// TwinCAT 3 PLC project Library_OOP
// Title: Library_OOP_Course
// Company: Course_OOP
// Author: Victor Duran -- Runtimevic
// ProjectVersion: 0.0.0.2
// Description: Library Couse OOP
// ProgramVersion: 3.1.4024.0
// libraries:
//   Library_OOP_Course, * (Course_OOP)
//   Tc2_Standard, * (Beckhoff Automation GmbH)
//   Tc2_System, * (Beckhoff Automation GmbH)
//   Tc3_Module, * (Beckhoff Automation GmbH)
// project tree:
//   Components/Cylinder/Interfaces/ I_AtHome.TcIO (not stored), I_AtWork.TcIO (not stored), I_MoveTo.TcIO (not stored)
//   FBs/ FB_FB_AXL_E_EC_DI8_DO8_M12_6P_BitMaps.TcPOU
//   FCs/ FC_Sum_int.TcPOU, FC_Word2Bools.TcPOU
//   / PlcTask.TcTTO
//   POUs/ MAIN.TcPOU
//   Project Information/ F_GetCompany.TcPOU, F_GetTitle.TcPOU, F_GetVersion.TcPOU
//   Units/DigitalInput/Class/ FB_DigitalInput.TcPOU (not stored)
//   Units/DigitalInput/Interface/ I_DigitalStatus.TcIO (not stored)
//   Units/DigitalOutput/Class/ FB_DigitalOutput.TcPOU (not stored)
//   Units/DigitalOutput/Interface/ I_DigitalOutput.TcIO (not stored)
//   Version/ Global_Version.TcGVL
// real-time tasks:
//   TASK PlcTask: cycle T#10ms, priority 20, ADS port 350

CONFIGURATION Library_OOP
    RESOURCE PLC ON TwinCAT3
        TASK PlcTask(INTERVAL := T#10ms, PRIORITY := 20);
        PROGRAM MAIN WITH PlcTask : MAIN;
    END_RESOURCE
END_CONFIGURATION

// ---- Version/Global_Version.TcGVL
{attribute 'TcGenerated'}
{attribute 'no-analysis'}
{attribute 'linkalways'}
// This function has been automatically generated from the project information.
VAR_GLOBAL CONSTANT
	{attribute 'const_non_replaced'}
	stLibVersion_Library_OOP_Course : ST_LibVersion := (iMajor := 0, iMinor := 0, iBuild := 0, iRevision := 2, nFlags := 1, sVersion := '0.0.0.2');
END_VAR

// ---- POUs/MAIN.TcPOU
PROGRAM MAIN
VAR
END_VAR

END_PROGRAM

// ---- FBs/FB_FB_AXL_E_EC_DI8_DO8_M12_6P_BitMaps.TcPOU
FUNCTION_BLOCK FB_FB_AXL_E_EC_DI8_DO8_M12_6P_BitMaps
VAR_INPUT
i_ModuleOut:ARRAY[1..8]OF BOOL;
END_VAR
VAR_OUTPUT
q_ModuleIn:ARRAY[1..8]OF BOOL;
q_DatosOK :BOOL;
END_VAR
VAR
DI1,DI2,DI3,DI4,DI5,DI6,Di7,DI8 AT %I*:BIT;
DO1,DO2,DO3,DO4,DO5,DO6,DO7,DO8 AT %Q*:BIT;
WcState AT %I*:BIT;
END_VAR

q_ModuleIn[1]:=DI1;
q_ModuleIn[2]:=DI2;
q_ModuleIn[3]:=DI3;
q_ModuleIn[4]:=DI4;
q_ModuleIn[5]:=DI5;
q_ModuleIn[6]:=DI6;
q_ModuleIn[7]:=DI7;
q_ModuleIn[8]:=DI8;

//Estado
q_DataOK:=NOT WcState;

//
DO1:=i_ModuleOut[1];
DO2:=i_ModuleOut[2];
DO3:=i_ModuleOut[3];
DO4:=i_ModuleOut[4];
DO5:=i_ModuleOut[5];
DO6:=i_ModuleOut[6];
DO7:=i_ModuleOut[7];
DO8:=i_ModuleOut[8];

END_FUNCTION_BLOCK

// ---- FCs/FC_Sum_int.TcPOU
FUNCTION FC_Sum_int : INT
VAR_INPUT
	operand1 : INT;
	operand2 : INT;
END_VAR
VAR
END_VAR


FC_Sum_int := operand1 + operand2

END_FUNCTION

// ---- FCs/FC_Word2Bools.TcPOU
FUNCTION FC_Word2Bools : ARRAY[0..7]OF BOOL
VAR_INPUT
	w16:WORD;
END_VAR
VAR
END_VAR

FC_Word2Bools[0]:=w16.0;
FC_Word2Bools[1]:=w16.1;
FC_Word2Bools[2]:=w16.2;
FC_Word2Bools[3]:=w16.3;
FC_Word2Bools[4]:=w16.4;
FC_Word2Bools[5]:=w16.5;
FC_Word2Bools[6]:=w16.6;
FC_Word2Bools[7]:=w16.7;

END_FUNCTION

// ---- Project Information/F_GetCompany.TcPOU
// This function has been automatically generated from the project information.
{attribute 'signature_flag' := '1073741824'}
{attribute 'TcGenerated'}
{attribute 'no-analysis'}
FUNCTION F_GetCompany : WSTRING
VAR_INPUT
	
END_VAR

F_GetCompany := "Course_OOP";

END_FUNCTION

// ---- Project Information/F_GetTitle.TcPOU
// This function has been automatically generated from the project information.
{attribute 'signature_flag' := '1073741824'}
{attribute 'TcGenerated'}
{attribute 'no-analysis'}
FUNCTION F_GetTitle : WSTRING
VAR_INPUT
	
END_VAR

F_GetTitle := "Library_OOP_Course";

END_FUNCTION

// ---- Project Information/F_GetVersion.TcPOU
// This function has been automatically generated from the project information.
{attribute 'signature_flag' := '1073741824'}
{attribute 'TcGenerated'}
{attribute 'no-analysis'}
FUNCTION F_GetVersion : ST_LibVersion
VAR_INPUT
	
END_VAR

F_GetVersion.iMajor := 0;
F_GetVersion.iMinor := 0;
F_GetVersion.iBuild := 0;
F_GetVersion.iRevision := 2;
F_GetVersion.sVersion := '0.0.0.2';
F_GetVersion.nFlags := 0;

END_FUNCTION
